// SIMATIC S7-200 project (STEP 7-Micro/WIN), CPU 224XP REL 02.01

SYMBOL_TABLE USER1
start            I0.0     // khoi dong he thong
stopp            I0.1     // dung he thong
s1               I0.2     // cam bien xe vao
s2               I0.3     // cam bien xe ra
k1               Q0.0     // bao day xe
END_SYMBOL_TABLE

ORGANIZATION_BLOCK MAIN:OB1
TITLE=PROGRAM COMMENTS
BEGIN
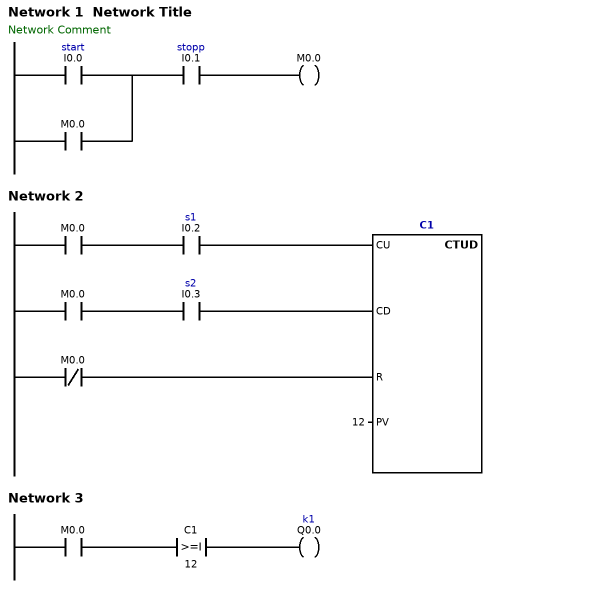
Network 1 // Network Title
// Network Comment
LD     start:I0.0
O      M0.0
A      stopp:I0.1
=      M0.0
Network 2
LD     M0.0
A      s1:I0.2
LD     M0.0
A      s2:I0.3
LDN    M0.0
CTUD   C1, 12
Network 3
LD     M0.0
AW>=   C1, 12
=      k1:Q0.0
END_ORGANIZATION_BLOCK
